// TIA Portal V21 export
TYPE "Std_VarGestAnalog"
   STRUCT
      In : Struct
         Ew : Word;
         ProfinetHwSubModule : HW_SUBMODULE;
         SondeDigitali : Struct
            Sonda_1Min : Bool;
            Sonda_2Med : Bool;
            Sonda_3Max : Bool;
         END_STRUCT;
         ActualValue_S7 : Real;
      END_STRUCT;
      Scalatura : Struct
         IngressoAnalogico : Real;
         OutMin : Real;
         OutMax : Real := 100.0;
         InMin : Real;
         InMax : Real := 27648.0;
         InMin_Leggi : Bool;
         InMax_Leggi : Bool;
      END_STRUCT;
      Prm : Struct
         K_TipoAnalogica : Int;   // 0 = IngressoAnalogicoPlc / 1 = ProfinetEndressHauser / 2 = SondeDigitali / 3 = ViaReteS7
         Inversione : Bool;   // 0 > 27648 / 27648 > 0
         PresetSoglia : Array[1..4] of Real;   // Questo valore indica il valore sopra il quale si setta la soglia di riferimento
         Isteresi : Array[1..4] of Real;   // Se si setta allarme sopra la soglia impostata si aspetta che scenda sotto soglia - isteresi per resettare
         RitSogliaOn { S7_SetPoint := 'True'} : Array[1..4] of "Std_stTimer";   // Tempo di ritardo On sulle soglie di allarme
         RitSogliaOf { S7_SetPoint := 'True'} : Array[1..4] of "Std_stTimer";   // Tempo di ritardo Of sulle soglie di allarme
         ModoSetAllarmeHmi : Array[1..4] of Bool;   // 0=SeSuperaSoglia 1=SeScendeSottoSoglia
         ModoResetAllarmeHmi : Array[1..4] of Bool;   // 0=Autoreset 1=TramitePulsanteReset
         UnitàMisura : "Std_UnitàDiMisura";
         FiltroUscita { S7_SetPoint := 'True'} : "Std_Lpf";   // Applico un filtro per rendere i valori più stabili
      END_STRUCT;
      Hmi : Struct
         ParatiaPresente : Bool;
         Simulazione : Struct
            Attiva : Bool;
            Valore : Int;   // 0 - 27648
            AbilitaTimeout : Bool := True;
            Timeout : "Std_stTimer";
         END_STRUCT;
         PopupSceltaVista : Struct
            TipoVista1 : Int;   // 0 Niente da visualizzare / 1 Analogica / 2 PID / 3 Totalizzatore / 4 Trend / 5 Paratia
            TipoVista2 : Int;   // 0 Niente da visualizzare / 1 Analogica / 2 PID / 3 Totalizzatore / 4 Trend / 5 Paratia
            TipoVista3 : Int;   // 0 Niente da visualizzare / 1 Analogica / 2 PID / 3 Totalizzatore / 4 Trend / 5 Paratia
            TipoVista4 : Int;   // 0 Niente da visualizzare / 1 Analogica / 2 PID / 3 Totalizzatore / 4 Trend / 5 Paratia
         END_STRUCT;
         UnitaMisura : Struct
            Converti : Bool;
            Calcola : Bool;
         END_STRUCT;
         NomeSoglia : Array[1..4] of String[18];
         AbilitaVistaSogliaHmi : Array[1..4] of Bool;   // 1=Rende la soglia modificabile da Hmi
      END_STRUCT;
      Dati : Struct
         PreOutSoglia : Array[1..4] of Bool;
      END_STRUCT;
      Allarmi : Struct
         "A" { S7_SetPoint := 'True'} : Array[0.."K_NumAllarmiPerAnalogiche"] of "Std_PrmAllarmeStd";
         WordHMI : Word;
      END_STRUCT;
      Out : Struct
         AnalogicaAttuale : "Std_ValoreConUm";
         SogliaMaxi : Bool;
         SogliaIntMax : Bool;
         SogliaIntMin : Bool;
         SogliaMini : Bool;
      END_STRUCT;
      Rif_Inc : Struct   // Serve per sapere chi legge e scrive
         K_Portata : Int;
         K_Pid_Uscita : Int;   // Il pid legge l'uscita del valore analogico
         K_Pid_Ingresso : Int;   // Il pid scrive il valore del'ingresso analogico
         K_Trend : Int;
         K_Paratia : Int;
         K_Analogica : Int;
      END_STRUCT;
   END_STRUCT;
   // // Prm.PresetSoglia[1] : Maxi
   // // Prm.PresetSoglia[2] : Intmax
   // // Prm.PresetSoglia[3] : Intmin
   // // Prm.PresetSoglia[4] : Mini
   // // Prm.Isteresi[1] : Maxi
   // // Prm.Isteresi[2] : Intmax
   // // Prm.Isteresi[3] : Intmin
   // // Prm.Isteresi[4] : Mini
   // // Prm.RitSogliaOn[1] : Maxi
   // // Prm.RitSogliaOn[2] : Intmax
   // // Prm.RitSogliaOn[3] : Intmin
   // // Prm.RitSogliaOn[4] : Mini
   // // Prm.RitSogliaOf[1] : Maxi
   // // Prm.RitSogliaOf[2] : Intmax
   // // Prm.RitSogliaOf[3] : Intmin
   // // Prm.RitSogliaOf[4] : Mini
   // // Prm.ModoSetAllarmeHmi[1] : Maxi
   // // Prm.ModoSetAllarmeHmi[2] : Intmax
   // // Prm.ModoSetAllarmeHmi[3] : Intmin
   // // Prm.ModoSetAllarmeHmi[4] : Mini
   // // Prm.ModoResetAllarmeHmi[1] : Maxi
   // // Prm.ModoResetAllarmeHmi[2] : Intmax
   // // Prm.ModoResetAllarmeHmi[3] : Intmin
   // // Prm.ModoResetAllarmeHmi[4] : Mini
   // Prm.UnitàMisura.In.UmCode := 40505;
   // Prm.UnitàMisura.Out.UmCode := 40505;
   // Prm.FiltroUscita.FattoreFiltro := 0.5;
   // Hmi.Simulazione.Timeout.Preset := 300.0;
   // Hmi.NomeSoglia[1] := 'massima';
   // Hmi.NomeSoglia[2] := 'intermedia massima';
   // Hmi.NomeSoglia[3] := 'intermedia minima';
   // Hmi.NomeSoglia[4] := 'minima';
   // Hmi.AbilitaVistaSogliaHmi[1] := True;   // Maxi
   // Hmi.AbilitaVistaSogliaHmi[2] := True;   // Intmax
   // Hmi.AbilitaVistaSogliaHmi[3] := True;   // Intmin
   // Hmi.AbilitaVistaSogliaHmi[4] := True;   // Mini
   // // Allarmi."A"[1] : Maxi
   // // Allarmi."A"[2] : IntMax
   // // Allarmi."A"[3] : IntMin
   // // Allarmi."A"[4] : Mini
   // // Allarmi."A"[5] : OutOfRange
END_TYPE
